INTERFACE ITF_MCHMIPrepareScreen_07_XX_Init

METHOD PUBLIC LinkDataHMI_07_XX : BOOL
VAR_INPUT
	refstData				: REFERENCE TO ST_MCHMIPrepareScreen_07_XX;
END_VAR
END_METHOD

END_INTERFACE

(* stored: Version 1.1.0.1
   Itf ITF_MCHMIPrepareScreen_07_XX_Init: Id {98f92c0f-1858-0b3d-209b-898ce385c756}
   Method LinkDataHMI_07_XX: Id {7df9f2e0-e302-03c3-1fef-fe05a6a0056f} *)
